PROGRAM P_Demo_FB_DALIV2QueryGroups
VAR
    fbFB_DALIV2QueryGroups        : FB_DALIV2QueryGroups;
    stCommandBuffer : ST_DALIV2CommandBuffer;

    bTrigger        : BOOL;
    nLampAddr        : BYTE := 0;

    wQueryGroups     : WORD;

    bBusy           : BOOL;
    bErr            : BOOL;
    nErrId          : UDINT;
END_VAR

// =============================================================================
// 场景：巡检读取 short addr 0 的 查询灯具完整组归属（合并 0-7 + 8-15 为 WORD）。
//
// 价值：HMI 实时显示 / 上线批量校验用。
//
// 验证步骤：
//   1. 通信 FB 跑起；编译；登录。
//   2. 在线 bTrigger 一次上升沿；等 bBusy 回 FALSE。
//   3. 观察 fbFB_DALIV2QueryGroups.wGroups 应为预期值（参考本 FB 文档 §4 描述）。
// =============================================================================
fbFB_DALIV2QueryGroups(
    bStart           := bTrigger,
    nAddr            := nLampAddr,
    eAddrType        := eDALIV2AddrTypeShort,
    eCommandPriority := eDALIV2CommandPriorityLow,
    stCommandBuffer  := stCommandBuffer
);

bBusy  := fbFB_DALIV2QueryGroups.bBusy;
bErr   := fbFB_DALIV2QueryGroups.bError;
nErrId := fbFB_DALIV2QueryGroups.nErrorId;

END_PROGRAM

(* stored: Version 1.1.0.1, ProductVersion 3.1.4024.5
   POU P_Demo_FB_DALIV2QueryGroups: Id {13f01014-c50b-54db-8b9d-a1ff5b2b767f}, SpecialFunc None *)
